// Deletes a generic's value.
FUNCTION F_Delete_Generic : BOOL
VAR_INPUT
	Source : REFERENCE TO T_Generic;
END_VAR
VAR
END_VAR

IF (NOT __ISVALIDREF(Source)) THEN RETURN; END_IF

CASE Tc2_System.F_CheckMemoryArea(Source.pValue, 1) OF
	Tc2_System.E_TcMemoryArea.Dynamic: __DELETE(Source.pValue);
ELSE
	Source.pValue := 0;
	END_CASE

Source.diSize := 0;
Source.TypeClass := T_Type.TYPE_NONE;

F_Delete_Generic := TRUE;

END_FUNCTION

(* stored: Version 1.1.0.1
   POU F_Delete_Generic: Id {911ffbfa-b462-0780-231b-8d2a2e64e20f}, SpecialFunc None *)
